ABB RobotStudio station: 6700_EGM_20220705-154103.rsstn

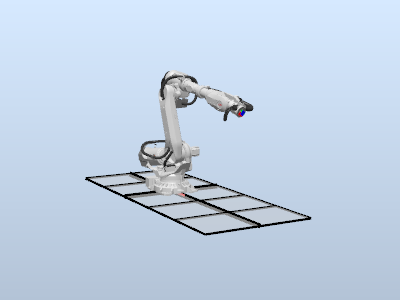
Station Station (saved by RobotStudio 22.2.9947.0)
Controller IRB6700_140_285_MH6
  mechanical unit ROB_1: IRB6700_140_285_MH6_04, 6 joints, base frame (0, 0, 0) mm
Layout (positions relative to the parent item):
  - IRB6700_140_285_MH6_04 [mechanism, from Robots\IRB6700_140_285_MH6_04.rslib] at (0, 0, 0) mm; joint values [0.1662, -0.0984, 0.3119, 0.044, 0.1458, -0.0272] (rad or m)
